// TwinCAT 3 PLC project ModbusRTU_lib
// Title: ModbusRTU_lib
// Company: Chua Siang Poh
// Author: Chua Siang Poh
// ProjectVersion: 1.0.0
// ProgramVersion: 3.1.4020.10
// libraries:
//   Tc2_ModbusRTU, * (Beckhoff Automation GmbH)
//   Tc2_Standard, * (Beckhoff Automation GmbH)
//   Tc2_System, * (Beckhoff Automation GmbH)
//   Tc3_Module, * (Beckhoff Automation GmbH)
// project tree:
//   MODBUS/ C_MODBUSMASTER.TcPOU, M_MODBUSSLAVE.TcPOU
//   MODBUS/DataType/ E_MODBUS_REGISTERTYPE.TcDUT, S_MODBUS_REGISTER.TcDUT
//   MODBUS/Functions/ F_TO_MODBUS_REGISTER.TcPOU
// (motion and I/O tree: see PLC project motion_library)
// real-time tasks:
//   TASK PlcTask: cycle T#10ms, priority 20, ADS port 350

// ---- MODBUS/DataType/E_MODBUS_REGISTERTYPE.TcDUT
{attribute 'qualified_only'}
{attribute 'strict'}
TYPE E_MODBUS_REGISTERTYPE :  
(
	E_MODBUS_INPUT := 0,
	E_MODBUS_OUTPUT := 16#800,
	E_MODBUS_MEMORY := 16#4000
) WORD;
END_TYPE

// ---- MODBUS/DataType/S_MODBUS_REGISTER.TcDUT
{attribute 'qualified_only'}
{attribute 'strict'}
TYPE S_MODBUS_REGISTER :
STRUCT
	REGISTER_SPACE	: E_MODBUS_REGISTERTYPE;
	REGISTER_OFFSET	: WORD;
	REGISTER_SIZE	: WORD;
END_STRUCT
END_TYPE

// ---- MODBUS/C_MODBUSMASTER.TcPOU
FUNCTION_BLOCK C_MODBUSMASTER
VAR_INPUT
END_VAR
VAR_OUTPUT
END_VAR
VAR
	_FBMASTER : ModbusRtuMaster_PcCOM;
END_VAR

METHOD HOLDING_REGISTER_READ : DINT
VAR_INPUT
	ID : USINT(1..247);
	
	REGISTER 		: S_MODBUS_REGISTER;
	
	buffer_ptr_out 	: PVOID;
	buffer_size 	: UINT;
END_VAR
_FBMASTER.UnitID := ID;
_FBMASTER.Quantity := REGISTER.REGISTER_SIZE;
_FBMASTER.MBAddr := F_TO_MODBUS_REGISTER(REGISTER);

_FBMASTER.Execute := TRUE;

_FBMASTER.pMemoryAddr := buffer_ptr_out;
_FBMASTER.cbLength := buffer_size;

_FBMASTER.Execute := TRUE;
_FBMASTER.ReadRegs();

IF _FBMASTER.Error THEN
	_FBMASTER.Execute := FALSE;
	_FBMASTER.ReadRegs();
	HOLDING_REGISTER_READ := 1;
	RETURN;
ELSIF NOT _FBMASTER.BUSY THEN
	_FBMASTER.Execute := FALSE;
	_FBMASTER.ReadRegs();
	HOLDING_REGISTER_READ := -1;
	RETURN;
ELSE
	HOLDING_REGISTER_READ := 0;
	RETURN;
END_IF
END_METHOD

METHOD HOLDING_REGISTER_WRITE : DINT
VAR_INPUT
	ID : USINT(1..247);
	
	REGISTER 		: S_MODBUS_REGISTER;
	
	buffer_ptr_out 	: PVOID;
	buffer_size 	: UINT;
END_VAR
_FBMASTER.UnitID := ID;

_FBMASTER.Quantity := REGISTER.REGISTER_SIZE;
_FBMASTER.MBAddr := F_TO_MODBUS_REGISTER(REGISTER);

_FBMASTER.pMemoryAddr := buffer_ptr_out;
_FBMASTER.cbLength := buffer_size;

_FBMASTER.Execute := TRUE;
_FBMASTER.WriteRegs();

IF _FBMASTER.Error THEN
	_FBMASTER.Execute := FALSE;
	_FBMASTER.WriteRegs();
	HOLDING_REGISTER_WRITE := 1;
	RETURN;
ELSIF NOT _FBMASTER.BUSY THEN
	_FBMASTER.Execute := FALSE;
	_FBMASTER.WriteRegs();
	HOLDING_REGISTER_WRITE := -1;
	RETURN;
ELSE
	HOLDING_REGISTER_WRITE := 0;
	RETURN;
END_IF
END_METHOD

END_FUNCTION_BLOCK

// ---- MODBUS/Functions/F_TO_MODBUS_REGISTER.TcPOU
FUNCTION F_TO_MODBUS_REGISTER : WORD
VAR_INPUT
	S_INFO : S_MODBUS_REGISTER;
END_VAR
VAR
	ADDRESS_SPACE : POINTER TO WORD;
END_VAR

ADDRESS_SPACE := ADR(S_INFO.REGISTER_SPACE);
F_TO_MODBUS_REGISTER := ADDRESS_SPACE^ + S_INFO.REGISTER_OFFSET;

END_FUNCTION

// ---- MODBUS/M_MODBUSSLAVE.TcPOU
FUNCTION_BLOCK M_MODBUSSLAVE
VAR_INPUT
END_VAR
VAR_OUTPUT
END_VAR
VAR
	_ENABLE : BOOL := FALSE;
	_FBSLAVE : ModbusRtuSlave_PcCOM;
	
	_MBINPUT 	: ARRAY[0..255] OF WORD;
	_MBOUTPUT 	: ARRAY[0..255] OF WORD;
	_MBMEMORY 	: ARRAY[0..255] OF WORD;
END_VAR

IF _ENABLE THEN
	_FBSLAVE(
		AdrInputs:= ADR(_MBINPUT), 
		SizeInputBytes:= SIZEOF(_MBINPUT), 
		AdrOutputs:= ADR(_MBOUTPUT), 
		SizeOutputBytes:= SIZEOF(_MBOUTPUT), 
		AdrMemory:= ADR(_MBMEMORY), 
		SizeMemoryBytes:= SIZEOF(_MBMEMORY), 
		ErrorId=> );
END_IF

PROPERTY ENABLE : BOOL
GET
ENABLE := _ENABLE;
END_GET
SET
_ENABLE := ENABLE;
END_SET
END_PROPERTY

METHOD FB_init : BOOL
VAR_INPUT
	bInitRetains : BOOL; // if TRUE, the retain variables are initialized (warm start / cold start)
	bInCopyCode : BOOL;  // if TRUE, the instance afterwards gets moved into the copy code (online change)

	DeviceID : UINT(1..247);
END_VAR
_FBSLAVE.UnitID := DeviceID;
END_METHOD

PROPERTY ID : UINT(1..247)
GET
ID := _FBSLAVE.UnitID;
END_GET
SET
_FBSLAVE.UnitID := ID;
END_SET
END_PROPERTY

PROPERTY INPUTS : POINTER TO BYTE
GET
INPUTS := ADR(_MBINPUT);
END_GET
END_PROPERTY

PROPERTY MEMORY : POINTER TO BYTE
GET
MEMORY := ADR(_MBMEMORY);
END_GET
END_PROPERTY

PROPERTY OUTPUTS : POINTER TO BYTE
GET
OUTPUTS := ADR(_MBOUTPUT);
END_GET
END_PROPERTY

END_FUNCTION_BLOCK
